PROGRAM MAIN
VAR
	 Delay1 : TON;
	 Delay2 : TON;
	 Delay3 : TON;
	 Delay4 : TON;
  
	XValueInt : INT;
	YValueInt :INT;
	
END_VAR

Delay1(IN:=TRUE, PT:=T#5S);

IF(Delay1.Q) THEN
   XValueInt := 3;
   YvalueInt := -2;
   
         Delay2(IN:=TRUE, PT:=T#5S);
         IF (Delay2.Q) THEN
			 
				XValueInt := -2;
	            YValueInt := 4;
	   
	                  Delay3(IN:=TRUE, PT:=T#5S);
					  
						IF (Delay3.Q) THEN
							XValueInt := 1;
	 					  YValueInt := 6;
						 			
										 Delay4(IN:=TRUE, PT:=T#5S);
					  
										IF (Delay4.Q) THEN
											XValueInt := -5;
	 									    YValueInt := -1;
											Delay1(IN:=FALSE, PT:=T#5S);
										END_IF
						END_IF
			END_IF
END_IF

END_PROGRAM

(* stored: Version 1.1.0.1, ProductVersion 3.1.4024.12
   POU MAIN: Id {1ab52c02-b4a6-415a-b3dd-b1834a2ea228}, SpecialFunc None *)
